RoboDK station: Anvendt_Robotteknikk_Lab3.rdk

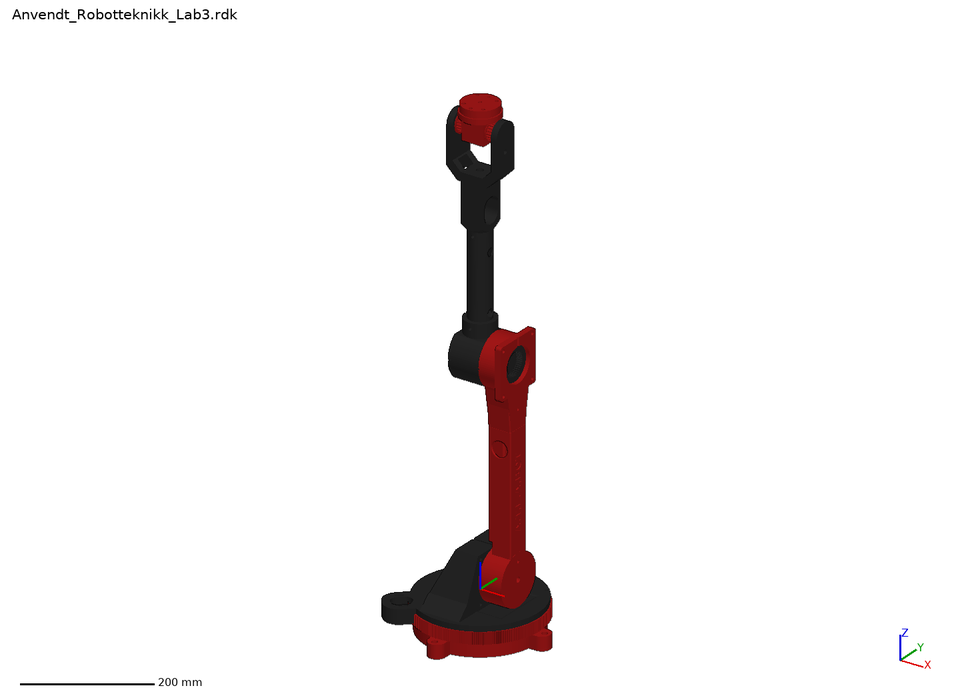
[picture v0: the station drawn from its stored meshes, robots at their saved joint values, targets as dots, program paths as lines]
Station Anvendt_Robotteknikk_Lab3 (saved by RoboDK 5.9.2). Poses are relative to the parent item; angles as X-Y-Z fixed-axis rotations.
  - frame Robot Frame at (0, 2000, 0) mm
    - robot ATLABOT: 6 axes
        modified DH rows (alpha deg, a mm, theta deg, d mm): 0, 0, 90, 35; -90, 0, 90, 0; 0, -355, 90, 0; -90, 0, 0, 375; 90, 0, 0, 0; -90, 0, 0, 40
        joint limits [-180, -90, -135, -360, -90, -180] to [180, 90, 135, 360, 90, 180]; home [0, 0, 0, 0, 0, 0]; saved at [0, 0, 0, 0, 0, 0]
  - Python program Prog1 (listed below)

--- Python program Prog1 ---
from time import sleep
from robodk.robolink import Robolink, ITEM_TYPE_TARGET, ITEM_TYPE_FRAME
RDK = Robolink()

from ATLABOT_library import RobotSerial
robot = RobotSerial('COM3')

t1 = RDK.Item('Target 1', ITEM_TYPE_TARGET)
t2 = RDK.Item('Target 2', ITEM_TYPE_TARGET)

f2 = RDK.Item('Frame 2', ITEM_TYPE_FRAME)


print("Test code")
robot.MoveJ(t2)
'''
print("")
sleep(0.5)
robot.MoveJ(f2)
print("")
sleep(0.5)
robot.home()
'''
